MOVJ C01770 VJ=0.78
MOVL C01771 V=8.0
MOVJ C01772 VJ=0.78
MOVJ C01773 VJ=0.78
MOVJ C01774 VJ=0.78
MOVL C01775 V=8.0
MOVJ C01776 VJ=0.78
MOVJ C01777 VJ=0.78
MOVJ C01778 VJ=0.78
MOVL C01779 V=8.0
MOVJ C01780 VJ=0.78
MOVJ C01781 VJ=0.78
MOVJ C01782 VJ=0.78
MOVL C01783 V=8.0
MOVJ C01784 VJ=0.78
MOVJ C01785 VJ=0.78
MOVJ C01786 VJ=0.78
MOVL C01787 V=8.0
MOVJ C01788 VJ=0.78
MOVJ C01789 VJ=0.78
MOVJ C01790 VJ=0.78
MOVL C01791 V=8.0
MOVJ C01792 VJ=0.78
MOVJ C01793 VJ=0.78
MOVJ C01794 VJ=0.78
MOVL C01795 V=8.0
MOVJ C01796 VJ=0.78
MOVJ C01797 VJ=0.78
MOVJ C01798 VJ=0.78
MOVL C01799 V=8.0
MOVJ C01800 VJ=0.78
MOVJ C01801 VJ=0.78
MOVJ C01802 VJ=0.78
MOVL C01803 V=8.0
MOVJ C01804 VJ=0.78
MOVJ C01805 VJ=0.78
MOVJ C01806 VJ=0.78
MOVL C01807 V=8.0
MOVJ C01808 VJ=0.78
MOVJ C01809 VJ=0.78
MOVJ C01810 VJ=0.78
MOVL C01811 V=8.0
MOVJ C01812 VJ=0.78
MOVJ C01813 VJ=0.78
MOVJ C01814 VJ=0.78
MOVL C01815 V=8.0
MOVJ C01816 VJ=0.78
MOVJ C01817 VJ=0.78
MOVJ C01818 VJ=0.78
MOVL C01819 V=8.0
MOVJ C01820 VJ=0.78
MOVJ C01821 VJ=0.78
MOVJ C01822 VJ=0.78
MOVL C01823 V=8.0
MOVJ C01824 VJ=0.78
MOVJ C01825 VJ=0.78
MOVJ C01826 VJ=0.78
MOVL C01827 V=8.0
MOVJ C01828 VJ=0.78
MOVJ C01829 VJ=0.78
MOVJ C01830 VJ=0.78
MOVL C01831 V=8.0
MOVJ C01832 VJ=0.78
MOVJ C01833 VJ=0.78
MOVJ C01834 VJ=0.78
MOVL C01835 V=8.0
MOVJ C01836 VJ=0.78
MOVJ C01837 VJ=0.78
MOVJ C01838 VJ=0.78
MOVL C01839 V=8.0
MOVJ C01840 VJ=0.78
MOVJ C01841 VJ=0.78
MOVJ C01842 VJ=0.78
MOVL C01843 V=8.0
MOVJ C01844 VJ=0.78
MOVJ C01845 VJ=0.78
MOVJ C01846 VJ=0.78
MOVL C01847 V=8.0
MOVJ C01848 VJ=0.78
MOVJ C01849 VJ=0.78
MOVJ C01850 VJ=0.78
MOVL C01851 V=8.0
MOVJ C01852 VJ=0.78
MOVJ C01853 VJ=0.78
MOVJ C01854 VJ=0.78
MOVL C01855 V=8.0
MOVJ C01856 VJ=0.78
MOVJ C01857 VJ=0.78
MOVJ C01858 VJ=0.78
MOVL C01859 V=8.0
MOVJ C01860 VJ=0.78
MOVJ C01861 VJ=0.78
MOVJ C01862 VJ=0.78
MOVL C01863 V=8.0
MOVJ C01864 VJ=0.78
MOVJ C01865 VJ=0.78
MOVJ C01866 VJ=0.78
MOVL C01867 V=8.0
MOVJ C01868 VJ=0.78
MOVJ C01869 VJ=0.78
MOVJ C01870 VJ=0.78
MOVL C01871 V=8.0
MOVJ C01872 VJ=0.78
MOVJ C01873 VJ=0.78
MOVJ C01874 VJ=0.78
MOVL C01875 V=8.0
MOVJ C01876 VJ=0.78
MOVJ C01877 VJ=0.78
MOVJ C01878 VJ=0.78
MOVL C01879 V=8.0
MOVJ C01880 VJ=0.78
MOVJ C01881 VJ=0.78
MOVJ C01882 VJ=0.78
MOVL C01883 V=8.0
MOVJ C01884 VJ=0.78
MOVJ C01885 VJ=0.78
MOVJ C01886 VJ=0.78
MOVL C01887 V=8.0
MOVJ C01888 VJ=0.78
MOVJ C01889 VJ=0.78
MOVJ C01890 VJ=0.78
MOVL C01891 V=8.0
MOVJ C01892 VJ=0.78
MOVJ C01893 VJ=0.78
MOVJ C01894 VJ=0.78
MOVL C01895 V=8.0
MOVJ C01896 VJ=0.78
MOVJ C01897 VJ=0.78
MOVJ C01898 VJ=0.78
MOVL C01899 V=8.0
MOVJ C01900 VJ=0.78
MOVJ C01901 VJ=0.78
MOVJ C01902 VJ=0.78
MOVL C01903 V=8.0
MOVJ C01904 VJ=0.78
MOVJ C01905 VJ=0.78
MOVJ C01906 VJ=0.78
MOVL C01907 V=8.0
MOVJ C01908 VJ=0.78
MOVJ C01909 VJ=0.78
MOVJ C01910 VJ=0.78
MOVL C01911 V=8.0
MOVJ C01912 VJ=0.78
MOVJ C01913 VJ=0.78
MOVJ C01914 VJ=0.78
MOVL C01915 V=8.0
MOVJ C01916 VJ=0.78
MOVJ C01917 VJ=0.78
MOVJ C01918 VJ=0.78
MOVL C01919 V=8.0
MOVJ C01920 VJ=0.78
MOVJ C01921 VJ=0.78
MOVJ C01922 VJ=0.78
MOVL C01923 V=8.0
MOVJ C01924 VJ=0.78
MOVJ C01925 VJ=0.78
MOVJ C01926 VJ=0.78
MOVL C01927 V=8.0
MOVJ C01928 VJ=0.78
MOVJ C01929 VJ=0.78
MOVJ C01930 VJ=0.78
MOVL C01931 V=8.0
MOVJ C01932 VJ=0.78
MOVJ C01933 VJ=0.78
MOVJ C01934 VJ=0.78
MOVL C01935 V=8.0
MOVJ C01936 VJ=0.78
MOVJ C01937 VJ=0.78
MOVJ C01938 VJ=0.78
MOVL C01939 V=8.0
MOVJ C01940 VJ=0.78
MOVJ C01941 VJ=0.78
MOVJ C01942 VJ=0.78
MOVL C01943 V=8.0
MOVJ C01944 VJ=0.78
MOVJ C01945 VJ=0.78
MOVJ C01946 VJ=0.78
MOVL C01947 V=8.0
MOVJ C01948 VJ=0.78
MOVJ C01949 VJ=0.78
MOVJ C01950 VJ=0.78
MOVL C01951 V=8.0
MOVJ C01952 VJ=0.78
MOVJ C01953 VJ=0.78
MOVJ C01954 VJ=0.78
MOVL C01955 V=8.0
MOVJ C01956 VJ=0.78
MOVJ C01957 VJ=0.78
MOVJ C01958 VJ=0.78
MOVL C01959 V=8.0
MOVJ C01960 VJ=0.78
MOVJ C01961 VJ=0.78
MOVJ C01962 VJ=0.78
MOVL C01963 V=8.0
MOVJ C01964 VJ=0.78
MOVJ C01965 VJ=0.78
MOVJ C01966 VJ=0.78
MOVL C01967 V=8.0
MOVJ C01968 VJ=0.78
MOVJ C01969 VJ=0.78
MOVJ C01970 VJ=0.78
MOVL C01971 V=8.0
MOVJ C01972 VJ=0.78
MOVJ C01973 VJ=0.78
MOVJ C01974 VJ=0.78
MOVL C01975 V=8.0
MOVJ C01976 VJ=0.78
MOVJ C01977 VJ=0.78
MOVJ C01978 VJ=0.78
MOVL C01979 V=8.0
MOVJ C01980 VJ=0.78
MOVJ C01981 VJ=0.78
MOVJ C01982 VJ=0.78
MOVL C01983 V=8.0
MOVJ C01984 VJ=0.78
MOVJ C01985 VJ=0.78
MOVJ C01986 VJ=0.78
MOVL C01987 V=8.0
MOVJ C01988 VJ=0.78
MOVJ C01989 VJ=0.78
MOVJ C01990 VJ=0.78
MOVL C01991 V=8.0
MOVJ C01992 VJ=0.78
MOVJ C01993 VJ=0.78
MOVJ C01994 VJ=0.78
MOVL C01995 V=8.0
MOVJ C01996 VJ=0.78
MOVJ C01997 VJ=0.78
MOVJ C01998 VJ=0.78
MOVL C01999 V=8.0
MOVJ C02000 VJ=0.78
MOVJ C02001 VJ=0.78
MOVJ C02002 VJ=0.78
MOVL C02003 V=8.0
MOVJ C02004 VJ=0.78
MOVJ C02005 VJ=0.78
MOVJ C02006 VJ=0.78
MOVL C02007 V=8.0
MOVJ C02008 VJ=0.78
MOVJ C02009 VJ=0.78
MOVJ C02010 VJ=0.78
MOVL C02011 V=8.0
MOVJ C02012 VJ=0.78
MOVJ C02013 VJ=0.78
MOVJ C02014 VJ=0.78
MOVL C02015 V=8.0
MOVJ C02016 VJ=0.78
MOVJ C02017 VJ=0.78
MOVJ C02018 VJ=0.78
MOVL C02019 V=8.0
MOVJ C02020 VJ=0.78
MOVJ C02021 VJ=0.78
MOVJ C02022 VJ=0.78
MOVL C02023 V=8.0
MOVJ C02024 VJ=0.78
MOVJ C02025 VJ=0.78
MOVJ C02026 VJ=0.78
MOVL C02027 V=8.0
MOVJ C02028 VJ=0.78
MOVJ C02029 VJ=0.78
MOVJ C02030 VJ=0.78
MOVL C02031 V=8.0
MOVJ C02032 VJ=0.78
MOVJ C02033 VJ=0.78
MOVJ C02034 VJ=0.78
MOVL C02035 V=8.0
MOVJ C02036 VJ=0.78
MOVJ C02037 VJ=0.78
MOVJ C02038 VJ=0.78
MOVL C02039 V=8.0
MOVJ C02040 VJ=0.78
MOVJ C02041 VJ=0.78
MOVJ C02042 VJ=0.78
MOVL C02043 V=8.0
MOVJ C02044 VJ=0.78
MOVJ C02045 VJ=0.78
MOVJ C02046 VJ=0.78
MOVL C02047 V=8.0
MOVJ C02048 VJ=0.78
MOVJ C02049 VJ=0.78
MOVJ C02050 VJ=0.78
MOVL C02051 V=8.0
MOVJ C02052 VJ=0.78
MOVJ C02053 VJ=0.78
MOVJ C02054 VJ=0.78
MOVL C02055 V=8.0
MOVJ C02056 VJ=0.78
MOVJ C02057 VJ=0.78
MOVJ C02058 VJ=0.78
MOVL C02059 V=8.0
MOVJ C02060 VJ=0.78
MOVJ C02061 VJ=0.78
MOVJ C02062 VJ=0.78
MOVL C02063 V=8.0
MOVJ C02064 VJ=0.78
MOVJ C02065 VJ=0.78
MOVJ C02066 VJ=0.78
MOVL C02067 V=8.0
MOVJ C02068 VJ=0.78
MOVJ C02069 VJ=0.78
MOVJ C02070 VJ=0.78
MOVL C02071 V=8.0
MOVJ C02072 VJ=0.78
MOVJ C02073 VJ=0.78
MOVJ C02074 VJ=0.78
MOVL C02075 V=8.0
MOVJ C02076 VJ=0.78
MOVJ C02077 VJ=0.78
MOVJ C02078 VJ=0.78
MOVL C02079 V=8.0
MOVJ C02080 VJ=0.78
MOVJ C02081 VJ=0.78
MOVJ C02082 VJ=0.78
MOVL C02083 V=8.0
MOVJ C02084 VJ=0.78
MOVJ C02085 VJ=0.78
MOVJ C02086 VJ=0.78
MOVL C02087 V=8.0
MOVJ C02088 VJ=0.78
MOVJ C02089 VJ=0.78
MOVJ C02090 VJ=0.78
MOVL C02091 V=8.0
MOVJ C02092 VJ=0.78
MOVJ C02093 VJ=0.78
MOVJ C02094 VJ=0.78
MOVL C02095 V=8.0
MOVJ C02096 VJ=0.78
MOVJ C02097 VJ=0.78
MOVJ C02098 VJ=0.78
MOVL C02099 V=8.0
MOVJ C02100 VJ=0.78
MOVJ C02101 VJ=0.78
MOVJ C02102 VJ=0.78
MOVL C02103 V=8.0
MOVJ C02104 VJ=0.78
MOVJ C02105 VJ=0.78
MOVJ C02106 VJ=0.78
MOVL C02107 V=8.0
MOVJ C02108 VJ=0.78
MOVJ C02109 VJ=0.78
MOVJ C02110 VJ=0.78
MOVL C02111 V=8.0
MOVJ C02112 VJ=0.78
MOVJ C02113 VJ=0.78
MOVJ C02114 VJ=0.78
MOVL C02115 V=8.0
MOVJ C02116 VJ=0.78
MOVJ C02117 VJ=0.78
MOVJ C02118 VJ=0.78
MOVL C02119 V=8.0
MOVJ C02120 VJ=0.78
MOVJ C02121 VJ=0.78
MOVJ C02122 VJ=0.78
MOVL C02123 V=8.0
MOVJ C02124 VJ=0.78
MOVJ C02125 VJ=0.78
MOVJ C02126 VJ=0.78
MOVL C02127 V=8.0
MOVJ C02128 VJ=0.78
MOVJ C02129 VJ=0.78
MOVJ C02130 VJ=0.78
MOVL C02131 V=8.0
MOVJ C02132 VJ=0.78
MOVJ C02133 VJ=0.78
MOVJ C02134 VJ=0.78
MOVL C02135 V=8.0
MOVJ C02136 VJ=0.78
MOVJ C02137 VJ=0.78
MOVJ C02138 VJ=0.78
MOVL C02139 V=8.0
MOVJ C02140 VJ=0.78
MOVJ C02141 VJ=0.78
MOVJ C02142 VJ=0.78
MOVL C02143 V=8.0
MOVJ C02144 VJ=0.78
MOVJ C02145 VJ=0.78
MOVJ C02146 VJ=0.78
MOVL C02147 V=8.0
MOVJ C02148 VJ=0.78
MOVJ C02149 VJ=0.78
MOVJ C02150 VJ=0.78
MOVL C02151 V=8.0
MOVJ C02152 VJ=0.78
MOVJ C02153 VJ=0.78
MOVJ C02154 VJ=0.78
MOVL C02155 V=8.0
MOVJ C02156 VJ=0.78
MOVJ C02157 VJ=0.78
MOVJ C02158 VJ=0.78
MOVL C02159 V=8.0
MOVJ C02160 VJ=0.78
MOVJ C02161 VJ=0.78
MOVJ C02162 VJ=0.78
MOVL C02163 V=8.0
MOVJ C02164 VJ=0.78
MOVJ C02165 VJ=0.78
MOVJ C02166 VJ=0.78
MOVL C02167 V=8.0
MOVJ C02168 VJ=0.78
MOVJ C02169 VJ=0.78
MOVJ C02170 VJ=0.78
MOVL C02171 V=8.0
MOVJ C02172 VJ=0.78
MOVJ C02173 VJ=0.78
MOVJ C02174 VJ=0.78
MOVL C02175 V=8.0
MOVJ C02176 VJ=0.78
MOVJ C02177 VJ=0.78
MOVJ C02178 VJ=0.78
MOVL C02179 V=8.0
MOVJ C02180 VJ=0.78
MOVJ C02181 VJ=0.78
MOVJ C02182 VJ=0.78
MOVL C02183 V=8.0
MOVJ C02184 VJ=0.78
MOVJ C02185 VJ=0.78
MOVJ C02186 VJ=0.78
MOVL C02187 V=8.0
MOVJ C02188 VJ=0.78
MOVJ C02189 VJ=0.78
MOVJ C02190 VJ=0.78
MOVL C02191 V=8.0
MOVJ C02192 VJ=0.78
MOVJ C02193 VJ=0.78
MOVJ C02194 VJ=0.78
MOVL C02195 V=8.0
MOVJ C02196 VJ=0.78
MOVJ C02197 VJ=0.78
MOVJ C02198 VJ=0.78
MOVL C02199 V=8.0
MOVJ C02200 VJ=0.78
MOVJ C02201 VJ=0.78
MOVJ C02202 VJ=0.78
MOVL C02203 V=8.0
MOVJ C02204 VJ=0.78
MOVJ C02205 VJ=0.78
MOVJ C02206 VJ=0.78
MOVL C02207 V=8.0
MOVJ C02208 VJ=0.78
MOVJ C02209 VJ=0.78
MOVJ C02210 VJ=0.78
MOVL C02211 V=8.0
MOVJ C02212 VJ=0.78
MOVJ C02213 VJ=0.78
MOVJ C02214 VJ=0.78
MOVL C02215 V=8.0
MOVJ C02216 VJ=0.78
MOVJ C02217 VJ=0.78
MOVJ C02218 VJ=0.78
MOVL C02219 V=8.0
MOVJ C02220 VJ=0.78
MOVJ C02221 VJ=0.78
MOVJ C02222 VJ=0.78
MOVL C02223 V=8.0
MOVJ C02224 VJ=0.78
MOVJ C02225 VJ=0.78
MOVJ C02226 VJ=0.78
MOVL C02227 V=8.0
MOVJ C02228 VJ=0.78
MOVJ C02229 VJ=0.78
MOVJ C02230 VJ=0.78
MOVL C02231 V=8.0
MOVJ C02232 VJ=0.78
MOVJ C02233 VJ=0.78
MOVJ C02234 VJ=0.78
MOVL C02235 V=8.0
MOVJ C02236 VJ=0.78
MOVJ C02237 VJ=0.78
MOVJ C02238 VJ=0.78
MOVL C02239 V=8.0
MOVJ C02240 VJ=0.78
MOVJ C02241 VJ=0.78
MOVJ C02242 VJ=0.78
MOVL C02243 V=8.0
MOVJ C02244 VJ=0.78
MOVJ C02245 VJ=0.78
MOVJ C02246 VJ=0.78
MOVL C02247 V=8.0
MOVJ C02248 VJ=0.78
MOVJ C02249 VJ=0.78
MOVJ C02250 VJ=0.78
MOVL C02251 V=8.0
MOVJ C02252 VJ=0.78
MOVJ C02253 VJ=0.78
MOVJ C02254 VJ=0.78
MOVL C02255 V=8.0
MOVJ C02256 VJ=0.78
MOVJ C02257 VJ=0.78
MOVJ C02258 VJ=0.78
MOVL C02259 V=8.0
MOVJ C02260 VJ=0.78
MOVJ C02261 VJ=0.78
MOVJ C02262 VJ=0.78
MOVL C02263 V=8.0
MOVJ C02264 VJ=0.78
MOVJ C02265 VJ=0.78
MOVJ C02266 VJ=0.78
MOVL C02267 V=8.0
MOVJ C02268 VJ=0.78
MOVJ C02269 VJ=0.78
MOVJ C02270 VJ=0.78
MOVL C02271 V=8.0
MOVJ C02272 VJ=0.78
MOVJ C02273 VJ=0.78
MOVJ C02274 VJ=0.78
MOVL C02275 V=8.0
MOVJ C02276 VJ=0.78
MOVJ C02277 VJ=0.78
MOVJ C02278 VJ=0.78
MOVL C02279 V=8.0
MOVJ C02280 VJ=0.78
MOVJ C02281 VJ=0.78
MOVJ C02282 VJ=0.78
MOVL C02283 V=8.0
MOVJ C02284 VJ=0.78
MOVJ C02285 VJ=0.78
MOVJ C02286 VJ=0.78
MOVL C02287 V=8.0
MOVJ C02288 VJ=0.78
MOVJ C02289 VJ=0.78
MOVJ C02290 VJ=0.78
MOVL C02291 V=8.0
MOVJ C02292 VJ=0.78
MOVJ C02293 VJ=0.78
MOVJ C02294 VJ=0.78
MOVL C02295 V=8.0
MOVJ C02296 VJ=0.78
MOVJ C02297 VJ=0.78
MOVJ C02298 VJ=0.78
MOVL C02299 V=8.0
MOVJ C02300 VJ=0.78
MOVJ C02301 VJ=0.78
MOVJ C02302 VJ=0.78
MOVL C02303 V=8.0
MOVJ C02304 VJ=0.78
MOVJ C02305 VJ=0.78
MOVJ C02306 VJ=0.78
MOVL C02307 V=8.0
MOVJ C02308 VJ=0.78
MOVJ C02309 VJ=0.78
MOVJ C02310 VJ=0.78
MOVL C02311 V=8.0
MOVJ C02312 VJ=0.78
MOVJ C02313 VJ=0.78
MOVJ C02314 VJ=0.78
MOVL C02315 V=8.0
MOVJ C02316 VJ=0.78
MOVJ C02317 VJ=0.78
MOVJ C02318 VJ=0.78
MOVL C02319 V=8.0
MOVJ C02320 VJ=0.78
MOVJ C02321 VJ=0.78
MOVJ C02322 VJ=0.78
MOVL C02323 V=8.0
MOVJ C02324 VJ=0.78
MOVJ C02325 VJ=0.78
MOVJ C02326 VJ=0.78
MOVL C02327 V=8.0
MOVJ C02328 VJ=0.78
MOVJ C02329 VJ=0.78
MOVJ C02330 VJ=0.78
MOVL C02331 V=8.0
MOVJ C02332 VJ=0.78
MOVJ C02333 VJ=0.78
MOVJ C02334 VJ=0.78
MOVL C02335 V=8.0
MOVJ C02336 VJ=0.78
MOVJ C02337 VJ=0.78
MOVJ C02338 VJ=0.78
MOVL C02339 V=8.0
MOVJ C02340 VJ=0.78
MOVJ C02341 VJ=0.78
MOVJ C02342 VJ=0.78
MOVL C02343 V=8.0
MOVJ C02344 VJ=0.78
MOVJ C02345 VJ=0.78
MOVJ C02346 VJ=0.78
MOVL C02347 V=8.0
MOVJ C02348 VJ=0.78
MOVJ C02349 VJ=0.78
MOVJ C02350 VJ=0.78
MOVL C02351 V=8.0
MOVJ C02352 VJ=0.78
MOVJ C02353 VJ=0.78
MOVJ C02354 VJ=0.78
MOVL C02355 V=8.0
MOVJ C02356 VJ=0.78
MOVJ C02357 VJ=0.78
MOVJ C02358 VJ=0.78
MOVL C02359 V=8.0
MOVJ C02360 VJ=0.78
MOVJ C02361 VJ=0.78
MOVJ C02362 VJ=0.78
MOVL C02363 V=8.0
MOVJ C02364 VJ=0.78
MOVJ C02365 VJ=0.78
MOVJ C02366 VJ=0.78
MOVL C02367 V=8.0
MOVJ C02368 VJ=0.78
MOVJ C02369 VJ=0.78
MOVJ C02370 VJ=0.78
MOVL C02371 V=8.0
MOVJ C02372 VJ=0.78
MOVJ C02373 VJ=0.78
MOVJ C02374 VJ=0.78
MOVL C02375 V=8.0
MOVJ C02376 VJ=0.78
MOVJ C02377 VJ=0.78
MOVJ C02378 VJ=0.78
MOVL C02379 V=8.0
MOVJ C02380 VJ=0.78
MOVJ C02381 VJ=0.78
MOVJ C02382 VJ=0.78
MOVL C02383 V=8.0
MOVJ C02384 VJ=0.78
MOVJ C02385 VJ=0.78
MOVJ C02386 VJ=0.78
MOVL C02387 V=8.0
MOVJ C02388 VJ=0.78
MOVJ C02389 VJ=0.78
MOVJ C02390 VJ=0.78
MOVL C02391 V=8.0
MOVJ C02392 VJ=0.78
MOVJ C02393 VJ=0.78
MOVJ C02394 VJ=0.78
MOVL C02395 V=8.0
MOVJ C02396 VJ=0.78
MOVJ C02397 VJ=0.78
MOVJ C02398 VJ=0.78
MOVL C02399 V=8.0
MOVJ C02400 VJ=0.78
MOVJ C02401 VJ=0.78
MOVJ C02402 VJ=0.78
MOVL C02403 V=8.0
MOVJ C02404 VJ=0.78
MOVJ C02405 VJ=0.78
MOVJ C02406 VJ=0.78
MOVL C02407 V=8.0
MOVJ C02408 VJ=0.78
MOVJ C02409 VJ=0.78
MOVJ C02410 VJ=0.78
MOVL C02411 V=8.0
MOVJ C02412 VJ=0.78
MOVJ C02413 VJ=0.78
MOVJ C02414 VJ=0.78
MOVL C02415 V=8.0
MOVJ C02416 VJ=0.78
MOVJ C02417 VJ=0.78
MOVJ C02418 VJ=0.78
MOVL C02419 V=8.0
MOVJ C02420 VJ=0.78
MOVJ C02421 VJ=0.78
MOVJ C02422 VJ=0.78
MOVL C02423 V=8.0
MOVJ C02424 VJ=0.78
MOVJ C02425 VJ=0.78
MOVJ C02426 VJ=0.78
MOVL C02427 V=8.0
MOVJ C02428 VJ=0.78
MOVJ C02429 VJ=0.78
MOVJ C02430 VJ=0.78
MOVL C02431 V=8.0
MOVJ C02432 VJ=0.78
MOVJ C02433 VJ=0.78
MOVJ C02434 VJ=0.78
MOVL C02435 V=8.0
MOVJ C02436 VJ=0.78
MOVJ C02437 VJ=0.78
MOVJ C02438 VJ=0.78
MOVL C02439 V=8.0
MOVJ C02440 VJ=0.78
MOVJ C02441 VJ=0.78
MOVJ C02442 VJ=0.78
MOVL C02443 V=8.0
MOVJ C02444 VJ=0.78
MOVJ C02445 VJ=0.78
MOVJ C02446 VJ=0.78
MOVL C02447 V=8.0
MOVJ C02448 VJ=0.78
MOVJ C02449 VJ=0.78
MOVJ C02450 VJ=0.78
MOVL C02451 V=8.0
MOVJ C02452 VJ=0.78
MOVJ C02453 VJ=0.78
MOVJ C02454 VJ=0.78
MOVL C02455 V=8.0
MOVJ C02456 VJ=0.78
MOVJ C02457 VJ=0.78
MOVJ C02458 VJ=0.78
MOVL C02459 V=8.0
MOVJ C02460 VJ=0.78
MOVJ C02461 VJ=0.78
MOVJ C02462 VJ=0.78
MOVL C02463 V=8.0
MOVJ C02464 VJ=0.78
MOVJ C02465 VJ=0.78
MOVJ C02466 VJ=0.78
MOVL C02467 V=8.0
MOVJ C02468 VJ=0.78
MOVJ C02469 VJ=0.78
MOVJ C02470 VJ=0.78
MOVL C02471 V=8.0
MOVJ C02472 VJ=0.78
MOVJ C02473 VJ=0.78
MOVJ C02474 VJ=0.78
MOVL C02475 V=8.0
MOVJ C02476 VJ=0.78
MOVJ C02477 VJ=0.78
MOVJ C02478 VJ=0.78
MOVL C02479 V=8.0
MOVJ C02480 VJ=0.78
MOVJ C02481 VJ=0.78
MOVJ C02482 VJ=0.78
MOVL C02483 V=8.0
MOVJ C02484 VJ=0.78
MOVJ C02485 VJ=0.78
MOVJ C02486 VJ=0.78
MOVL C02487 V=8.0
MOVJ C02488 VJ=0.78
MOVJ C02489 VJ=0.78
MOVJ C02490 VJ=0.78
MOVL C02491 V=8.0
MOVJ C02492 VJ=0.78
MOVJ C02493 VJ=0.78
MOVJ C02494 VJ=0.78
MOVL C02495 V=8.0
MOVJ C02496 VJ=0.78
MOVJ C02497 VJ=0.78
MOVJ C02498 VJ=0.78
MOVL C02499 V=8.0
MOVJ C02500 VJ=0.78
MOVJ C02501 VJ=0.78
MOVJ C02502 VJ=0.78
MOVL C02503 V=8.0
MOVJ C02504 VJ=0.78
MOVJ C02505 VJ=0.78
MOVJ C02506 VJ=0.78
MOVL C02507 V=8.0
MOVJ C02508 VJ=0.78
MOVJ C02509 VJ=0.78
MOVJ C02510 VJ=0.78
MOVL C02511 V=8.0
MOVJ C02512 VJ=0.78
MOVJ C02513 VJ=0.78
MOVJ C02514 VJ=0.78
MOVL C02515 V=8.0
MOVJ C02516 VJ=0.78
MOVJ C02517 VJ=0.78
MOVJ C02518 VJ=0.78
MOVL C02519 V=8.0
MOVJ C02520 VJ=0.78
MOVJ C02521 VJ=0.78
MOVJ C02522 VJ=0.78
MOVL C02523 V=8.0
MOVJ C02524 VJ=0.78
MOVJ C02525 VJ=0.78
MOVJ C02526 VJ=0.78
MOVL C02527 V=8.0
MOVJ C02528 VJ=0.78
MOVJ C02529 VJ=0.78
MOVJ C02530 VJ=0.78
MOVL C02531 V=8.0
MOVJ C02532 VJ=0.78
MOVJ C02533 VJ=0.78
MOVJ C02534 VJ=0.78
MOVL C02535 V=8.0
MOVJ C02536 VJ=0.78
MOVJ C02537 VJ=0.78
MOVJ C02538 VJ=0.78
MOVL C02539 V=8.0
MOVJ C02540 VJ=0.78
MOVJ C02541 VJ=0.78
MOVJ C02542 VJ=0.78
MOVL C02543 V=8.0
MOVJ C02544 VJ=0.78
MOVJ C02545 VJ=0.78
MOVJ C02546 VJ=0.78
MOVL C02547 V=8.0
MOVJ C02548 VJ=0.78
MOVJ C02549 VJ=0.78
MOVJ C02550 VJ=0.78
MOVL C02551 V=8.0
MOVJ C02552 VJ=0.78
MOVJ C02553 VJ=0.78
MOVJ C02554 VJ=0.78
MOVL C02555 V=8.0
MOVJ C02556 VJ=0.78
MOVJ C02557 VJ=0.78
MOVJ C02558 VJ=0.78
MOVL C02559 V=8.0
MOVJ C02560 VJ=0.78
MOVJ C02561 VJ=0.78
MOVJ C02562 VJ=0.78
MOVL C02563 V=8.0
MOVJ C02564 VJ=0.78
MOVJ C02565 VJ=0.78
MOVJ C02566 VJ=0.78
MOVL C02567 V=8.0
MOVJ C02568 VJ=0.78
MOVJ C02569 VJ=0.78
MOVJ C02570 VJ=0.78
MOVL C02571 V=8.0
MOVJ C02572 VJ=0.78
MOVJ C02573 VJ=0.78
MOVJ C02574 VJ=0.78
MOVL C02575 V=8.0
MOVJ C02576 VJ=0.78
MOVJ C02577 VJ=0.78
MOVJ C02578 VJ=0.78
MOVL C02579 V=8.0
MOVJ C02580 VJ=0.78
MOVJ C02581 VJ=0.78
MOVJ C02582 VJ=0.78
MOVL C02583 V=8.0
MOVJ C02584 VJ=0.78
MOVJ C02585 VJ=0.78
MOVJ C02586 VJ=0.78
MOVL C02587 V=8.0
MOVJ C02588 VJ=0.78
MOVJ C02589 VJ=0.78
MOVJ C02590 VJ=0.78
MOVL C02591 V=8.0
MOVJ C02592 VJ=0.78
MOVJ C02593 VJ=0.78
MOVJ C02594 VJ=0.78
MOVL C02595 V=8.0
MOVJ C02596 VJ=0.78
MOVJ C02597 VJ=0.78
MOVJ C02598 VJ=0.78
MOVL C02599 V=8.0
MOVJ C02600 VJ=0.78
MOVJ C02601 VJ=0.78
MOVJ C02602 VJ=0.78
MOVL C02603 V=8.0
MOVJ C02604 VJ=0.78
MOVJ C02605 VJ=0.78
MOVJ C02606 VJ=0.78
MOVL C02607 V=8.0
MOVJ C02608 VJ=0.78
MOVJ C02609 VJ=0.78
MOVJ C02610 VJ=0.78
MOVL C02611 V=8.0
MOVJ C02612 VJ=0.78
MOVJ C02613 VJ=0.78
MOVJ C02614 VJ=0.78
MOVL C02615 V=8.0
MOVJ C02616 VJ=0.78
MOVJ C02617 VJ=0.78
MOVJ C02618 VJ=0.78
MOVL C02619 V=8.0
MOVJ C02620 VJ=0.78
MOVJ C02621 VJ=0.78
MOVJ C02622 VJ=0.78
MOVL C02623 V=8.0
MOVJ C02624 VJ=0.78
MOVJ C02625 VJ=0.78
MOVJ C02626 VJ=0.78
MOVL C02627 V=8.0
MOVJ C02628 VJ=0.78
MOVJ C02629 VJ=0.78
MOVJ C02630 VJ=0.78
MOVL C02631 V=8.0
MOVJ C02632 VJ=0.78
MOVJ C02633 VJ=0.78
MOVJ C02634 VJ=0.78
MOVL C02635 V=8.0
MOVJ C02636 VJ=0.78
MOVJ C02637 VJ=0.78
MOVJ C02638 VJ=0.78
MOVL C02639 V=8.0
MOVJ C02640 VJ=0.78
MOVJ C02641 VJ=0.78
MOVJ C02642 VJ=0.78
MOVL C02643 V=8.0
MOVJ C02644 VJ=0.78
MOVJ C02645 VJ=0.78
MOVJ C02646 VJ=0.78
MOVL C02647 V=8.0
MOVJ C02648 VJ=0.78
MOVJ C02649 VJ=0.78
MOVJ C02650 VJ=0.78
MOVL C02651 V=8.0
MOVJ C02652 VJ=0.78
MOVJ C02653 VJ=0.78
MOVJ C02654 VJ=0.78
MOVL C02655 V=8.0
MOVJ C02656 VJ=0.78
MOVJ C02657 VJ=0.78
MOVJ C02658 VJ=0.78
MOVL C02659 V=8.0
MOVJ C02660 VJ=0.78
MOVJ C02661 VJ=0.78
MOVJ C02662 VJ=0.78
MOVL C02663 V=8.0
MOVJ C02664 VJ=0.78
MOVJ C02665 VJ=0.78
MOVJ C02666 VJ=0.78
MOVL C02667 V=8.0
MOVJ C02668 VJ=0.78
MOVJ C02669 VJ=0.78
MOVJ C02670 VJ=0.78
MOVL C02671 V=8.0
MOVJ C02672 VJ=0.78
MOVJ C02673 VJ=0.78
MOVJ C02674 VJ=0.78
MOVL C02675 V=8.0
MOVJ C02676 VJ=0.78
MOVJ C02677 VJ=0.78
MOVJ C02678 VJ=0.78
MOVL C02679 V=8.0
MOVJ C02680 VJ=0.78
MOVJ C02681 VJ=0.78
MOVJ C02682 VJ=0.78
MOVL C02683 V=8.0
MOVJ C02684 VJ=0.78
MOVJ C02685 VJ=0.78
MOVJ C02686 VJ=0.78
MOVL C02687 V=8.0
MOVJ C02688 VJ=0.78
MOVJ C02689 VJ=0.78
MOVJ C02690 VJ=0.78
MOVL C02691 V=8.0
MOVJ C02692 VJ=0.78
MOVJ C02693 VJ=0.78
MOVJ C02694 VJ=0.78
MOVL C02695 V=8.0
MOVJ C02696 VJ=0.78
MOVJ C02697 VJ=0.78
MOVJ C02698 VJ=0.78
MOVL C02699 V=8.0
MOVJ C02700 VJ=0.78
MOVJ C02701 VJ=0.78
MOVJ C02702 VJ=0.78
MOVL C02703 V=8.0
MOVJ C02704 VJ=0.78
MOVJ C02705 VJ=0.78
MOVJ C02706 VJ=0.78
MOVL C02707 V=8.0
MOVJ C02708 VJ=0.78
MOVJ C02709 VJ=0.78
MOVJ C02710 VJ=0.78
MOVL C02711 V=8.0
MOVJ C02712 VJ=0.78
MOVJ C02713 VJ=0.78
MOVJ C02714 VJ=0.78
MOVL C02715 V=8.0
MOVJ C02716 VJ=0.78
MOVJ C02717 VJ=0.78
MOVJ C02718 VJ=0.78
MOVL C02719 V=8.0
MOVJ C02720 VJ=0.78
MOVJ C02721 VJ=0.78
MOVJ C02722 VJ=0.78
MOVL C02723 V=8.0
MOVJ C02724 VJ=0.78
MOVJ C02725 VJ=0.78
MOVJ C02726 VJ=0.78
MOVL C02727 V=8.0
MOVJ C02728 VJ=0.78
MOVJ C02729 VJ=0.78
MOVJ C02730 VJ=0.78
MOVL C02731 V=8.0
MOVJ C02732 VJ=0.78
MOVJ C02733 VJ=0.78
MOVJ C02734 VJ=0.78
MOVL C02735 V=8.0
MOVJ C02736 VJ=0.78
MOVJ C02737 VJ=0.78
MOVJ C02738 VJ=0.78
MOVL C02739 V=8.0
MOVJ C02740 VJ=0.78
MOVJ C02741 VJ=0.78
MOVJ C02742 VJ=0.78
MOVL C02743 V=8.0
MOVJ C02744 VJ=0.78
MOVJ C02745 VJ=0.78
MOVJ C02746 VJ=0.78
MOVL C02747 V=8.0
MOVJ C02748 VJ=0.78
MOVJ C02749 VJ=0.78
MOVJ C02750 VJ=0.78
MOVL C02751 V=8.0
MOVJ C02752 VJ=0.78
MOVJ C02753 VJ=0.78
MOVJ C02754 VJ=0.78
MOVL C02755 V=8.0
MOVJ C02756 VJ=0.78
MOVJ C02757 VJ=0.78
MOVJ C02758 VJ=0.78
MOVL C02759 V=8.0
MOVJ C02760 VJ=0.78
MOVJ C02761 VJ=0.78
MOVJ C02762 VJ=0.78
MOVL C02763 V=8.0
MOVJ C02764 VJ=0.78
MOVJ C02765 VJ=0.78
MOVJ C02766 VJ=0.78
MOVL C02767 V=8.0
MOVJ C02768 VJ=0.78
MOVJ C02769 VJ=0.78
MOVJ C02770 VJ=0.78
MOVL C02771 V=8.0
MOVJ C02772 VJ=0.78
MOVJ C02773 VJ=0.78
MOVJ C02774 VJ=0.78
MOVL C02775 V=8.0
MOVJ C02776 VJ=0.78
MOVJ C02777 VJ=0.78
MOVJ C02778 VJ=0.78
MOVL C02779 V=8.0
MOVJ C02780 VJ=0.78
MOVJ C02781 VJ=0.78
MOVJ C02782 VJ=0.78
MOVL C02783 V=8.0
MOVJ C02784 VJ=0.78
MOVJ C02785 VJ=0.78
MOVJ C02786 VJ=0.78
MOVL C02787 V=8.0
MOVJ C02788 VJ=0.78
MOVJ C02789 VJ=0.78
MOVJ C02790 VJ=0.78
MOVL C02791 V=8.0
MOVJ C02792 VJ=0.78
MOVJ C02793 VJ=0.78
MOVJ C02794 VJ=0.78
MOVL C02795 V=8.0
MOVJ C02796 VJ=0.78
MOVJ C02797 VJ=0.78
MOVJ C02798 VJ=0.78
MOVL C02799 V=8.0
MOVJ C02800 VJ=0.78
MOVJ C02801 VJ=0.78
MOVJ C02802 VJ=0.78
MOVL C02803 V=8.0
MOVJ C02804 VJ=0.78
MOVJ C02805 VJ=0.78
MOVJ C02806 VJ=0.78
MOVL C02807 V=8.0
MOVJ C02808 VJ=0.78
MOVJ C02809 VJ=0.78
MOVJ C02810 VJ=0.78
MOVL C02811 V=8.0
MOVJ C02812 VJ=0.78
MOVJ C02813 VJ=0.78
MOVJ C02814 VJ=0.78
MOVL C02815 V=8.0
MOVJ C02816 VJ=0.78
MOVJ C02817 VJ=0.78
MOVJ C02818 VJ=0.78
MOVL C02819 V=8.0
MOVJ C02820 VJ=0.78
MOVJ C02821 VJ=0.78
MOVJ C02822 VJ=0.78
MOVL C02823 V=8.0
MOVJ C02824 VJ=0.78
MOVJ C02825 VJ=0.78
MOVJ C02826 VJ=0.78
MOVL C02827 V=8.0
MOVJ C02828 VJ=0.78
MOVJ C02829 VJ=0.78
MOVJ C02830 VJ=0.78
MOVL C02831 V=8.0
MOVJ C02832 VJ=0.78
MOVJ C02833 VJ=0.78
MOVJ C02834 VJ=0.78
MOVL C02835 V=8.0
MOVJ C02836 VJ=0.78
MOVJ C02837 VJ=0.78
MOVJ C02838 VJ=0.78
MOVL C02839 V=8.0
MOVJ C02840 VJ=0.78
MOVJ C02841 VJ=0.78
MOVJ C02842 VJ=0.78
MOVL C02843 V=8.0
MOVJ C02844 VJ=0.78
MOVJ C02845 VJ=0.78
MOVJ C02846 VJ=0.78
MOVL C02847 V=8.0
MOVJ C02848 VJ=0.78
MOVJ C02849 VJ=0.78
MOVJ C02850 VJ=0.78
MOVL C02851 V=8.0
MOVJ C02852 VJ=0.78
MOVJ C02853 VJ=0.78
MOVJ C02854 VJ=0.78
MOVL C02855 V=8.0
MOVJ C02856 VJ=0.78
MOVJ C02857 VJ=0.78
MOVJ C02858 VJ=0.78
MOVL C02859 V=8.0
MOVJ C02860 VJ=0.78
MOVJ C02861 VJ=0.78
MOVJ C02862 VJ=0.78
MOVL C02863 V=8.0
MOVJ C02864 VJ=0.78
MOVJ C02865 VJ=0.78
MOVJ C02866 VJ=0.78
MOVL C02867 V=8.0
MOVJ C02868 VJ=0.78
MOVJ C02869 VJ=0.78
MOVJ C02870 VJ=0.78
MOVL C02871 V=8.0
MOVJ C02872 VJ=0.78
MOVJ C02873 VJ=0.78
MOVJ C02874 VJ=0.78
MOVL C02875 V=8.0
MOVJ C02876 VJ=0.78
MOVJ C02877 VJ=0.78
MOVJ C02878 VJ=0.78
MOVL C02879 V=8.0
MOVJ C02880 VJ=0.78
MOVJ C02881 VJ=0.78
MOVJ C02882 VJ=0.78
MOVL C02883 V=8.0
MOVJ C02884 VJ=0.78
MOVJ C02885 VJ=0.78
MOVJ C02886 VJ=0.78
MOVL C02887 V=8.0
MOVJ C02888 VJ=0.78
MOVJ C02889 VJ=0.78
MOVJ C02890 VJ=0.78
MOVL C02891 V=8.0
MOVJ C02892 VJ=0.78
MOVJ C02893 VJ=0.78
MOVJ C02894 VJ=0.78
MOVL C02895 V=8.0
MOVJ C02896 VJ=0.78
MOVJ C02897 VJ=0.78
MOVJ C02898 VJ=0.78
MOVL C02899 V=8.0
MOVJ C02900 VJ=0.78
MOVJ C02901 VJ=0.78
MOVJ C02902 VJ=0.78
MOVL C02903 V=8.0
MOVJ C02904 VJ=0.78
MOVJ C02905 VJ=0.78
MOVJ C02906 VJ=0.78
MOVL C02907 V=8.0
MOVJ C02908 VJ=0.78
MOVJ C02909 VJ=0.78
MOVJ C02910 VJ=0.78
MOVL C02911 V=8.0
MOVJ C02912 VJ=0.78
MOVJ C02913 VJ=0.78
MOVJ C02914 VJ=0.78
MOVL C02915 V=8.0
MOVJ C02916 VJ=0.78
MOVJ C02917 VJ=0.78
MOVJ C02918 VJ=0.78
MOVL C02919 V=8.0
MOVJ C02920 VJ=0.78
MOVJ C02921 VJ=0.78
MOVJ C02922 VJ=0.78
MOVL C02923 V=8.0
MOVJ C02924 VJ=0.78
MOVJ C02925 VJ=0.78
MOVJ C02926 VJ=0.78
MOVL C02927 V=8.0
MOVJ C02928 VJ=0.78
MOVJ C02929 VJ=0.78
MOVJ C02930 VJ=0.78
MOVL C02931 V=8.0
MOVJ C02932 VJ=0.78
MOVJ C02933 VJ=0.78
MOVJ C02934 VJ=0.78
MOVL C02935 V=8.0
MOVJ C02936 VJ=0.78
MOVJ C02937 VJ=0.78
MOVJ C02938 VJ=0.78
MOVL C02939 V=8.0
MOVJ C02940 VJ=0.78
MOVJ C02941 VJ=0.78
MOVJ C02942 VJ=0.78
MOVL C02943 V=8.0
MOVJ C02944 VJ=0.78
MOVJ C02945 VJ=0.78
MOVJ C02946 VJ=0.78
MOVL C02947 V=8.0
MOVJ C02948 VJ=0.78
MOVJ C02949 VJ=0.78
MOVJ C02950 VJ=0.78
MOVL C02951 V=8.0
MOVJ C02952 VJ=0.78
MOVJ C02953 VJ=0.78
MOVJ C02954 VJ=0.78
MOVL C02955 V=8.0
MOVJ C02956 VJ=0.78
MOVJ C02957 VJ=0.78
MOVJ C02958 VJ=0.78
MOVL C02959 V=8.0
MOVJ C02960 VJ=0.78
MOVJ C02961 VJ=0.78
MOVJ C02962 VJ=0.78
MOVL C02963 V=8.0
MOVJ C02964 VJ=0.78
MOVJ C02965 VJ=0.78
MOVJ C02966 VJ=0.78
MOVL C02967 V=8.0
MOVJ C02968 VJ=0.78
MOVJ C02969 VJ=0.78
MOVJ C02970 VJ=0.78
MOVL C02971 V=8.0
MOVJ C02972 VJ=0.78
MOVJ C02973 VJ=0.78
MOVJ C02974 VJ=0.78
MOVL C02975 V=8.0
MOVJ C02976 VJ=0.78
MOVJ C02977 VJ=0.78
MOVJ C02978 VJ=0.78
MOVL C02979 V=8.0
MOVJ C02980 VJ=0.78
MOVJ C02981 VJ=0.78
MOVJ C02982 VJ=0.78
MOVL C02983 V=8.0
MOVJ C02984 VJ=0.78
MOVJ C02985 VJ=0.78
MOVJ C02986 VJ=0.78
MOVL C02987 V=8.0
MOVJ C02988 VJ=0.78
MOVJ C02989 VJ=0.78
MOVJ C02990 VJ=0.78
MOVL C02991 V=8.0
MOVJ C02992 VJ=0.78
MOVJ C02993 VJ=0.78
MOVJ C02994 VJ=0.78
MOVL C02995 V=8.0
MOVJ C02996 VJ=0.78
MOVJ C02997 VJ=0.78
MOVJ C02998 VJ=0.78
MOVL C02999 V=8.0
MOVJ C03000 VJ=0.78
MOVJ C03001 VJ=0.78
MOVJ C03002 VJ=0.78
MOVL C03003 V=8.0
MOVJ C03004 VJ=0.78
MOVJ C03005 VJ=0.78
MOVJ C03006 VJ=0.78
MOVL C03007 V=8.0
MOVJ C03008 VJ=0.78
MOVJ C03009 VJ=0.78
MOVJ C03010 VJ=0.78
MOVL C03011 V=8.0
MOVJ C03012 VJ=0.78
MOVJ C03013 VJ=0.78
MOVJ C03014 VJ=0.78
MOVL C03015 V=8.0
MOVJ C03016 VJ=0.78
MOVJ C03017 VJ=0.78
MOVJ C03018 VJ=0.78
MOVL C03019 V=8.0
MOVJ C03020 VJ=0.78
MOVJ C03021 VJ=0.78
MOVJ C03022 VJ=0.78
MOVL C03023 V=8.0
MOVJ C03024 VJ=0.78
MOVJ C03025 VJ=0.78
MOVJ C03026 VJ=0.78
MOVL C03027 V=8.0
MOVJ C03028 VJ=0.78
MOVJ C03029 VJ=0.78
MOVJ C03030 VJ=0.78
MOVL C03031 V=8.0
MOVJ C03032 VJ=0.78
MOVJ C03033 VJ=0.78
MOVJ C03034 VJ=0.78
MOVL C03035 V=8.0
MOVJ C03036 VJ=0.78
MOVJ C03037 VJ=0.78
MOVJ C03038 VJ=0.78
MOVL C03039 V=8.0
MOVJ C03040 VJ=0.78
MOVJ C03041 VJ=0.78
MOVJ C03042 VJ=0.78
MOVL C03043 V=8.0
MOVJ C03044 VJ=0.78
MOVJ C03045 VJ=0.78
MOVJ C03046 VJ=0.78
MOVL C03047 V=8.0
MOVJ C03048 VJ=0.78
MOVJ C03049 VJ=0.78
MOVJ C03050 VJ=0.78
MOVL C03051 V=8.0
MOVJ C03052 VJ=0.78
MOVJ C03053 VJ=0.78
MOVJ C03054 VJ=0.78
MOVL C03055 V=8.0
MOVJ C03056 VJ=0.78
MOVJ C03057 VJ=0.78
MOVJ C03058 VJ=0.78
MOVL C03059 V=8.0
MOVJ C03060 VJ=0.78
MOVJ C03061 VJ=0.78
MOVJ C03062 VJ=0.78
MOVL C03063 V=8.0
MOVJ C03064 VJ=0.78
MOVJ C03065 VJ=0.78
MOVJ C03066 VJ=0.78
MOVL C03067 V=8.0
MOVJ C03068 VJ=0.78
MOVJ C03069 VJ=0.78
MOVJ C03070 VJ=0.78
MOVL C03071 V=8.0
MOVJ C03072 VJ=0.78
MOVJ C03073 VJ=0.78
MOVJ C03074 VJ=0.78
MOVL C03075 V=8.0
MOVJ C03076 VJ=0.78
MOVJ C03077 VJ=0.78
MOVJ C03078 VJ=0.78
MOVL C03079 V=8.0
MOVJ C03080 VJ=0.78
MOVJ C03081 VJ=0.78
MOVJ C03082 VJ=0.78
MOVL C03083 V=8.0
MOVJ C03084 VJ=0.78
MOVJ C03085 VJ=0.78
MOVJ C03086 VJ=0.78
MOVL C03087 V=8.0
MOVJ C03088 VJ=0.78
MOVJ C03089 VJ=0.78
MOVJ C03090 VJ=0.78
MOVL C03091 V=8.0
MOVJ C03092 VJ=0.78
MOVJ C03093 VJ=0.78
MOVJ C03094 VJ=0.78
MOVL C03095 V=8.0
MOVJ C03096 VJ=0.78
MOVJ C03097 VJ=0.78
MOVJ C03098 VJ=0.78
MOVL C03099 V=8.0
MOVJ C03100 VJ=0.78
MOVJ C03101 VJ=0.78
MOVJ C03102 VJ=0.78
MOVL C03103 V=8.0
MOVJ C03104 VJ=0.78
MOVJ C03105 VJ=0.78
MOVJ C03106 VJ=0.78
MOVL C03107 V=8.0
MOVJ C03108 VJ=0.78
MOVJ C03109 VJ=0.78
MOVJ C03110 VJ=0.78
MOVL C03111 V=8.0
MOVJ C03112 VJ=0.78
MOVJ C03113 VJ=0.78
MOVJ C03114 VJ=0.78
MOVL C03115 V=8.0
MOVJ C03116 VJ=0.78
MOVJ C03117 VJ=0.78
MOVJ C03118 VJ=0.78
MOVL C03119 V=8.0
MOVJ C03120 VJ=0.78
MOVJ C03121 VJ=0.78
MOVJ C03122 VJ=0.78
MOVL C03123 V=8.0
MOVJ C03124 VJ=0.78
MOVJ C03125 VJ=0.78
MOVJ C03126 VJ=0.78
MOVL C03127 V=8.0
MOVJ C03128 VJ=0.78
MOVJ C03129 VJ=0.78
MOVJ C03130 VJ=0.78
MOVL C03131 V=8.0
MOVJ C03132 VJ=0.78
MOVJ C03133 VJ=0.78
MOVJ C03134 VJ=0.78
MOVL C03135 V=8.0
MOVJ C03136 VJ=0.78
MOVJ C03137 VJ=0.78
MOVJ C03138 VJ=0.78
MOVL C03139 V=8.0
MOVJ C03140 VJ=0.78
MOVJ C03141 VJ=0.78
MOVJ C03142 VJ=0.78
MOVL C03143 V=8.0
MOVJ C03144 VJ=0.78
MOVJ C03145 VJ=0.78
MOVJ C03146 VJ=0.78
MOVL C03147 V=8.0
MOVJ C03148 VJ=0.78
MOVJ C03149 VJ=0.78
MOVJ C03150 VJ=0.78
MOVL C03151 V=8.0
MOVJ C03152 VJ=0.78
MOVJ C03153 VJ=0.78
MOVJ C03154 VJ=0.78
MOVL C03155 V=8.0
MOVJ C03156 VJ=0.78
MOVJ C03157 VJ=0.78
MOVJ C03158 VJ=0.78
MOVL C03159 V=8.0
MOVJ C03160 VJ=0.78
MOVJ C03161 VJ=0.78
MOVJ C03162 VJ=0.78
MOVL C03163 V=8.0
MOVJ C03164 VJ=0.78
MOVJ C03165 VJ=0.78
MOVJ C03166 VJ=0.78
MOVL C03167 V=8.0
MOVJ C03168 VJ=0.78
MOVJ C03169 VJ=0.78
MOVJ C03170 VJ=0.78
MOVL C03171 V=8.0
MOVJ C03172 VJ=0.78
MOVJ C03173 VJ=0.78
MOVJ C03174 VJ=0.78
MOVL C03175 V=8.0
MOVJ C03176 VJ=0.78
MOVJ C03177 VJ=0.78
MOVJ C03178 VJ=0.78
MOVL C03179 V=8.0
MOVJ C03180 VJ=0.78
MOVJ C03181 VJ=0.78
MOVJ C03182 VJ=0.78
MOVL C03183 V=8.0
MOVJ C03184 VJ=0.78
MOVJ C03185 VJ=0.78
MOVJ C03186 VJ=0.78
MOVL C03187 V=8.0
MOVJ C03188 VJ=0.78
MOVJ C03189 VJ=0.78
MOVJ C03190 VJ=0.78
MOVL C03191 V=8.0
MOVJ C03192 VJ=0.78
MOVJ C03193 VJ=0.78
MOVJ C03194 VJ=0.78
MOVL C03195 V=8.0
MOVJ C03196 VJ=0.78
MOVJ C03197 VJ=0.78
MOVJ C03198 VJ=0.78
MOVL C03199 V=8.0
MOVJ C03200 VJ=0.78
MOVJ C03201 VJ=0.78
MOVJ C03202 VJ=0.78
MOVL C03203 V=8.0
MOVJ C03204 VJ=0.78
MOVJ C03205 VJ=0.78
MOVJ C03206 VJ=0.78
MOVL C03207 V=8.0
MOVJ C03208 VJ=0.78
MOVJ C03209 VJ=0.78
MOVJ C03210 VJ=0.78
MOVL C03211 V=8.0
MOVJ C03212 VJ=0.78
MOVJ C03213 VJ=0.78
MOVJ C03214 VJ=0.78
MOVL C03215 V=8.0
MOVJ C03216 VJ=0.78
MOVJ C03217 VJ=0.78
MOVJ C03218 VJ=0.78
MOVL C03219 V=8.0
MOVJ C03220 VJ=0.78
MOVJ C03221 VJ=0.78
MOVJ C03222 VJ=0.78
MOVL C03223 V=8.0
MOVJ C03224 VJ=0.78
MOVJ C03225 VJ=0.78
MOVJ C03226 VJ=0.78
MOVL C03227 V=8.0
MOVJ C03228 VJ=0.78
MOVJ C03229 VJ=0.78
MOVJ C03230 VJ=0.78
MOVL C03231 V=8.0
MOVJ C03232 VJ=0.78
MOVJ C03233 VJ=0.78
MOVJ C03234 VJ=0.78
MOVL C03235 V=8.0
MOVJ C03236 VJ=0.78
MOVJ C03237 VJ=0.78
MOVJ C03238 VJ=0.78
MOVL C03239 V=8.0
MOVJ C03240 VJ=0.78
MOVJ C03241 VJ=0.78
MOVJ C03242 VJ=0.78
MOVL C03243 V=8.0
MOVJ C03244 VJ=0.78
MOVJ C03245 VJ=0.78
MOVJ C03246 VJ=0.78
MOVL C03247 V=8.0
MOVJ C03248 VJ=0.78
MOVJ C03249 VJ=0.78
MOVJ C03250 VJ=0.78
MOVL C03251 V=8.0
MOVJ C03252 VJ=0.78
MOVJ C03253 VJ=0.78
MOVJ C03254 VJ=0.78
MOVL C03255 V=8.0
MOVJ C03256 VJ=0.78
MOVJ C03257 VJ=0.78
MOVJ C03258 VJ=0.78
MOVL C03259 V=8.0
MOVJ C03260 VJ=0.78
MOVJ C03261 VJ=0.78
MOVJ C03262 VJ=0.78
MOVL C03263 V=8.0
MOVJ C03264 VJ=0.78
MOVJ C03265 VJ=0.78
MOVJ C03266 VJ=0.78
MOVL C03267 V=8.0
MOVJ C03268 VJ=0.78
MOVJ C03269 VJ=0.78
MOVJ C03270 VJ=0.78
MOVL C03271 V=8.0
MOVJ C03272 VJ=0.78
MOVJ C03273 VJ=0.78
MOVJ C03274 VJ=0.78
MOVL C03275 V=8.0
MOVJ C03276 VJ=0.78
MOVJ C03277 VJ=0.78
MOVJ C03278 VJ=0.78
MOVL C03279 V=8.0
MOVJ C03280 VJ=0.78
MOVJ C03281 VJ=0.78
MOVJ C03282 VJ=0.78
MOVL C03283 V=8.0
MOVJ C03284 VJ=0.78
MOVJ C03285 VJ=0.78
MOVJ C03286 VJ=0.78
MOVL C03287 V=8.0
MOVJ C03288 VJ=0.78
MOVJ C03289 VJ=0.78
MOVJ C03290 VJ=0.78
MOVL C03291 V=8.0
MOVJ C03292 VJ=0.78
MOVJ C03293 VJ=0.78
MOVJ C03294 VJ=0.78
MOVL C03295 V=8.0
MOVJ C03296 VJ=0.78
MOVJ C03297 VJ=0.78
MOVJ C03298 VJ=0.78
MOVL C03299 V=8.0
MOVJ C03300 VJ=0.78
MOVJ C03301 VJ=0.78
MOVJ C03302 VJ=0.78
MOVL C03303 V=8.0
MOVJ C03304 VJ=0.78
MOVJ C03305 VJ=0.78
MOVJ C03306 VJ=0.78
MOVL C03307 V=8.0
MOVJ C03308 VJ=0.78
MOVJ C03309 VJ=0.78
MOVJ C03310 VJ=0.78
MOVL C03311 V=8.0
MOVJ C03312 VJ=0.78
MOVJ C03313 VJ=0.78
MOVJ C03314 VJ=0.78
MOVL C03315 V=8.0
MOVJ C03316 VJ=0.78
MOVJ C03317 VJ=0.78
MOVJ C03318 VJ=0.78
MOVL C03319 V=8.0
MOVJ C03320 VJ=0.78
MOVJ C03321 VJ=0.78
MOVJ C03322 VJ=0.78
MOVL C03323 V=8.0
MOVJ C03324 VJ=0.78
MOVJ C03325 VJ=0.78
MOVJ C03326 VJ=0.78
MOVL C03327 V=8.0
MOVJ C03328 VJ=0.78
MOVJ C03329 VJ=0.78
MOVJ C03330 VJ=0.78
MOVL C03331 V=8.0
MOVJ C03332 VJ=0.78
MOVJ C03333 VJ=0.78
MOVJ C03334 VJ=0.78
MOVL C03335 V=8.0
MOVJ C03336 VJ=0.78
MOVJ C03337 VJ=0.78
MOVJ C03338 VJ=0.78
MOVL C03339 V=8.0
MOVJ C03340 VJ=0.78
MOVJ C03341 VJ=0.78
MOVJ C03342 VJ=0.78
MOVL C03343 V=8.0
MOVJ C03344 VJ=0.78
MOVJ C03345 VJ=0.78
MOVJ C03346 VJ=0.78
MOVL C03347 V=8.0
MOVJ C03348 VJ=0.78
MOVJ C03349 VJ=0.78
MOVJ C03350 VJ=0.78
MOVL C03351 V=8.0
MOVJ C03352 VJ=0.78
MOVJ C03353 VJ=0.78
MOVJ C03354 VJ=0.78
MOVL C03355 V=8.0
MOVJ C03356 VJ=0.78
MOVJ C03357 VJ=0.78
MOVJ C03358 VJ=0.78
MOVL C03359 V=8.0
MOVJ C03360 VJ=0.78
MOVJ C03361 VJ=0.78
MOVJ C03362 VJ=0.78
MOVL C03363 V=8.0
MOVJ C03364 VJ=0.78
MOVJ C03365 VJ=0.78
MOVJ C03366 VJ=0.78
MOVL C03367 V=8.0
MOVJ C03368 VJ=0.78
MOVJ C03369 VJ=0.78
MOVJ C03370 VJ=0.78
MOVL C03371 V=8.0
MOVJ C03372 VJ=0.78
MOVJ C03373 VJ=0.78
MOVJ C03374 VJ=0.78
MOVL C03375 V=8.0
MOVJ C03376 VJ=0.78
MOVJ C03377 VJ=0.78
MOVJ C03378 VJ=0.78
MOVL C03379 V=8.0
MOVJ C03380 VJ=0.78
MOVJ C03381 VJ=0.78
MOVJ C03382 VJ=0.78
MOVL C03383 V=8.0
MOVJ C03384 VJ=0.78
MOVJ C03385 VJ=0.78
MOVJ C03386 VJ=0.78
MOVL C03387 V=8.0
MOVJ C03388 VJ=0.78
MOVJ C03389 VJ=0.78
MOVJ C03390 VJ=0.78
MOVL C03391 V=8.0
MOVJ C03392 VJ=0.78
MOVJ C03393 VJ=0.78
MOVJ C03394 VJ=0.78
MOVL C03395 V=8.0
MOVJ C03396 VJ=0.78
MOVJ C03397 VJ=0.78
MOVJ C03398 VJ=0.78
MOVL C03399 V=8.0
MOVJ C03400 VJ=0.78
MOVJ C03401 VJ=0.78
MOVJ C03402 VJ=0.78
MOVL C03403 V=8.0
MOVJ C03404 VJ=0.78
MOVJ C03405 VJ=0.78
MOVJ C03406 VJ=0.78
MOVL C03407 V=8.0
MOVJ C03408 VJ=0.78
MOVJ C03409 VJ=0.78
MOVJ C03410 VJ=0.78
MOVL C03411 V=8.0
MOVJ C03412 VJ=0.78
MOVJ C03413 VJ=0.78
MOVJ C03414 VJ=0.78
MOVL C03415 V=8.0
MOVJ C03416 VJ=0.78
MOVJ C03417 VJ=0.78
MOVJ C03418 VJ=0.78
MOVL C03419 V=8.0
MOVJ C03420 VJ=0.78
MOVJ C03421 VJ=0.78
MOVJ C03422 VJ=0.78
MOVL C03423 V=8.0
MOVJ C03424 VJ=0.78
MOVJ C03425 VJ=0.78
MOVJ C03426 VJ=0.78
MOVL C03427 V=8.0
MOVJ C03428 VJ=0.78
MOVJ C03429 VJ=0.78
MOVJ C03430 VJ=0.78
MOVL C03431 V=8.0
MOVJ C03432 VJ=0.78
MOVJ C03433 VJ=0.78
MOVJ C03434 VJ=0.78
MOVL C03435 V=8.0
MOVJ C03436 VJ=0.78
MOVJ C03437 VJ=0.78
MOVJ C03438 VJ=0.78
MOVL C03439 V=8.0
MOVJ C03440 VJ=0.78
MOVJ C03441 VJ=0.78
MOVJ C03442 VJ=0.78
MOVL C03443 V=8.0
MOVJ C03444 VJ=0.78
MOVJ C03445 VJ=0.78
MOVJ C03446 VJ=0.78
MOVL C03447 V=8.0
MOVJ C03448 VJ=0.78
MOVJ C03449 VJ=0.78
MOVJ C03450 VJ=0.78
MOVL C03451 V=8.0
MOVJ C03452 VJ=0.78
MOVJ C03453 VJ=0.78
MOVJ C03454 VJ=0.78
MOVL C03455 V=8.0
MOVJ C03456 VJ=0.78
MOVJ C03457 VJ=0.78
MOVJ C03458 VJ=0.78
MOVL C03459 V=8.0
MOVJ C03460 VJ=0.78
MOVJ C03461 VJ=0.78
MOVJ C03462 VJ=0.78
MOVL C03463 V=8.0
MOVJ C03464 VJ=0.78
MOVJ C03465 VJ=0.78
MOVJ C03466 VJ=0.78
MOVL C03467 V=8.0
MOVJ C03468 VJ=0.78
MOVJ C03469 VJ=0.78
MOVJ C03470 VJ=0.78
MOVL C03471 V=8.0
MOVJ C03472 VJ=0.78
MOVJ C03473 VJ=0.78
MOVJ C03474 VJ=0.78
MOVL C03475 V=8.0
MOVJ C03476 VJ=0.78
MOVJ C03477 VJ=0.78
MOVJ C03478 VJ=0.78
MOVL C03479 V=8.0
MOVJ C03480 VJ=0.78
MOVJ C03481 VJ=0.78
MOVJ C03482 VJ=0.78
MOVL C03483 V=8.0
MOVJ C03484 VJ=0.78
MOVJ C03485 VJ=0.78
MOVJ C03486 VJ=0.78
MOVL C03487 V=8.0
MOVJ C03488 VJ=0.78
MOVJ C03489 VJ=0.78
MOVJ C03490 VJ=0.78
MOVL C03491 V=8.0
MOVJ C03492 VJ=0.78
MOVJ C03493 VJ=0.78
MOVJ C03494 VJ=0.78
MOVL C03495 V=8.0
MOVJ C03496 VJ=0.78
MOVJ C03497 VJ=0.78
MOVJ C03498 VJ=0.78
MOVL C03499 V=8.0
MOVJ C03500 VJ=0.78
MOVJ C03501 VJ=0.78
MOVJ C03502 VJ=0.78
MOVL C03503 V=8.0
MOVJ C03504 VJ=0.78
MOVJ C03505 VJ=0.78
MOVJ C03506 VJ=0.78
MOVL C03507 V=8.0
MOVJ C03508 VJ=0.78
MOVJ C03509 VJ=0.78
MOVJ C03510 VJ=0.78
MOVL C03511 V=8.0
MOVJ C03512 VJ=0.78
MOVJ C03513 VJ=0.78
MOVJ C03514 VJ=0.78
MOVL C03515 V=8.0
MOVJ C03516 VJ=0.78
MOVJ C03517 VJ=0.78
MOVJ C03518 VJ=0.78
MOVL C03519 V=8.0
MOVJ C03520 VJ=0.78
MOVJ C03521 VJ=0.78
MOVJ C03522 VJ=0.78
MOVL C03523 V=8.0
MOVJ C03524 VJ=0.78
MOVJ C03525 VJ=0.78
MOVJ C03526 VJ=0.78
MOVL C03527 V=8.0
MOVJ C03528 VJ=0.78
MOVJ C03529 VJ=0.78
MOVJ C03530 VJ=0.78
MOVL C03531 V=8.0
MOVJ C03532 VJ=0.78
MOVJ C03533 VJ=0.78
MOVJ C03534 VJ=0.78
MOVL C03535 V=8.0
MOVJ C03536 VJ=0.78
MOVJ C03537 VJ=0.78
MOVJ C03538 VJ=0.78
MOVL C03539 V=8.0
MOVJ C03540 VJ=0.78
MOVJ C03541 VJ=0.78
MOVJ C03542 VJ=0.78
MOVL C03543 V=8.0
MOVJ C03544 VJ=0.78
MOVJ C03545 VJ=0.78
MOVJ C03546 VJ=0.78
MOVL C03547 V=8.0
MOVJ C03548 VJ=0.78
MOVJ C03549 VJ=0.78
MOVJ C03550 VJ=0.78
MOVL C03551 V=8.0
MOVJ C03552 VJ=0.78
MOVJ C03553 VJ=0.78
MOVJ C03554 VJ=0.78
MOVL C03555 V=8.0
MOVJ C03556 VJ=0.78
MOVJ C03557 VJ=0.78
MOVJ C03558 VJ=0.78
MOVL C03559 V=8.0
MOVJ C03560 VJ=0.78
MOVJ C03561 VJ=0.78
MOVJ C03562 VJ=0.78
MOVL C03563 V=8.0
MOVJ C03564 VJ=0.78
MOVJ C03565 VJ=0.78
MOVJ C03566 VJ=0.78
MOVL C03567 V=8.0
MOVJ C03568 VJ=0.78
MOVJ C03569 VJ=0.78
MOVJ C03570 VJ=0.78
MOVL C03571 V=8.0
MOVJ C03572 VJ=0.78
MOVJ C03573 VJ=0.78
MOVJ C03574 VJ=0.78
MOVL C03575 V=8.0
MOVJ C03576 VJ=0.78
MOVJ C03577 VJ=0.78
MOVJ C03578 VJ=0.78
MOVL C03579 V=8.0
MOVJ C03580 VJ=0.78
MOVJ C03581 VJ=0.78
MOVJ C03582 VJ=0.78
MOVL C03583 V=8.0
MOVJ C03584 VJ=0.78
MOVJ C03585 VJ=0.78
MOVJ C03586 VJ=0.78
MOVL C03587 V=8.0
MOVJ C03588 VJ=0.78
MOVJ C03589 VJ=0.78
MOVJ C03590 VJ=0.78
MOVL C03591 V=8.0
MOVJ C03592 VJ=0.78
MOVJ C03593 VJ=0.78
MOVJ C03594 VJ=0.78
MOVL C03595 V=8.0
MOVJ C03596 VJ=0.78
MOVJ C03597 VJ=0.78
MOVJ C03598 VJ=0.78
MOVL C03599 V=8.0
MOVJ C03600 VJ=0.78
MOVJ C03601 VJ=0.78
MOVJ C03602 VJ=0.78
MOVL C03603 V=8.0
MOVJ C03604 VJ=0.78
MOVJ C03605 VJ=0.78
MOVJ C03606 VJ=0.78
MOVL C03607 V=8.0
MOVJ C03608 VJ=0.78
MOVJ C03609 VJ=0.78
MOVJ C03610 VJ=0.78
MOVL C03611 V=8.0
MOVJ C03612 VJ=0.78
MOVJ C03613 VJ=0.78
MOVJ C03614 VJ=0.78
MOVL C03615 V=8.0
MOVJ C03616 VJ=0.78
MOVJ C03617 VJ=0.78
MOVJ C03618 VJ=0.78
MOVL C03619 V=8.0
MOVJ C03620 VJ=0.78
MOVJ C03621 VJ=0.78
MOVJ C03622 VJ=0.78
MOVL C03623 V=8.0
MOVJ C03624 VJ=0.78
MOVJ C03625 VJ=0.78
MOVJ C03626 VJ=0.78
MOVL C03627 V=8.0
MOVJ C03628 VJ=0.78
MOVJ C03629 VJ=0.78
MOVJ C03630 VJ=0.78
MOVL C03631 V=8.0
MOVJ C03632 VJ=0.78
MOVJ C03633 VJ=0.78
MOVJ C03634 VJ=0.78
MOVL C03635 V=8.0
MOVJ C03636 VJ=0.78
MOVJ C03637 VJ=0.78
MOVJ C03638 VJ=0.78
MOVL C03639 V=8.0
MOVJ C03640 VJ=0.78
MOVJ C03641 VJ=0.78
MOVJ C03642 VJ=0.78
MOVL C03643 V=8.0
MOVJ C03644 VJ=0.78
MOVJ C03645 VJ=0.78
MOVJ C03646 VJ=0.78
MOVL C03647 V=8.0
MOVJ C03648 VJ=0.78
MOVJ C03649 VJ=0.78
MOVJ C03650 VJ=0.78
MOVL C03651 V=8.0
MOVJ C03652 VJ=0.78
MOVJ C03653 VJ=0.78
MOVJ C03654 VJ=0.78
MOVL C03655 V=8.0
MOVJ C03656 VJ=0.78
MOVJ C03657 VJ=0.78
MOVJ C03658 VJ=0.78
MOVL C03659 V=8.0
MOVJ C03660 VJ=0.78
MOVJ C03661 VJ=0.78
MOVJ C03662 VJ=0.78
MOVL C03663 V=8.0
MOVJ C03664 VJ=0.78
MOVJ C03665 VJ=0.78
MOVJ C03666 VJ=0.78
MOVL C03667 V=8.0
MOVJ C03668 VJ=0.78
MOVJ C03669 VJ=0.78
MOVJ C03670 VJ=0.78
MOVL C03671 V=8.0
MOVJ C03672 VJ=0.78
MOVJ C03673 VJ=0.78
MOVJ C03674 VJ=0.78
MOVL C03675 V=8.0
MOVJ C03676 VJ=0.78
MOVJ C03677 VJ=0.78
MOVJ C03678 VJ=0.78
MOVL C03679 V=8.0
MOVJ C03680 VJ=0.78
MOVJ C03681 VJ=0.78
MOVJ C03682 VJ=0.78
MOVL C03683 V=8.0
MOVJ C03684 VJ=0.78
MOVJ C03685 VJ=0.78
MOVJ C03686 VJ=0.78
MOVL C03687 V=8.0
MOVJ C03688 VJ=0.78
MOVJ C03689 VJ=0.78
MOVJ C03690 VJ=0.78
MOVL C03691 V=8.0
MOVJ C03692 VJ=0.78
MOVJ C03693 VJ=0.78
MOVJ C03694 VJ=0.78
MOVL C03695 V=8.0
MOVJ C03696 VJ=0.78
MOVJ C03697 VJ=0.78
MOVJ C03698 VJ=0.78
MOVL C03699 V=8.0
MOVJ C03700 VJ=0.78
MOVJ C03701 VJ=0.78
MOVJ C03702 VJ=0.78
MOVL C03703 V=8.0
MOVJ C03704 VJ=0.78
MOVJ C03705 VJ=0.78
MOVJ C03706 VJ=0.78
MOVL C03707 V=8.0
MOVJ C03708 VJ=0.78
MOVJ C03709 VJ=0.78
MOVJ C03710 VJ=0.78
MOVL C03711 V=8.0
MOVJ C03712 VJ=0.78
MOVJ C03713 VJ=0.78
MOVJ C03714 VJ=0.78
MOVL C03715 V=8.0
MOVJ C03716 VJ=0.78
MOVJ C03717 VJ=0.78
MOVJ C03718 VJ=0.78
MOVL C03719 V=8.0
MOVJ C03720 VJ=0.78
MOVJ C03721 VJ=0.78
MOVJ C03722 VJ=0.78
MOVL C03723 V=8.0
MOVJ C03724 VJ=0.78
MOVJ C03725 VJ=0.78
MOVJ C03726 VJ=0.78
MOVL C03727 V=8.0
MOVJ C03728 VJ=0.78
MOVJ C03729 VJ=0.78
MOVJ C03730 VJ=0.78
MOVL C03731 V=8.0
MOVJ C03732 VJ=0.78
MOVJ C03733 VJ=0.78
MOVJ C03734 VJ=0.78
MOVL C03735 V=8.0
MOVJ C03736 VJ=0.78
MOVJ C03737 VJ=0.78
MOVJ C03738 VJ=0.78
MOVL C03739 V=8.0
MOVJ C03740 VJ=0.78
MOVJ C03741 VJ=0.78
MOVJ C03742 VJ=0.78
MOVL C03743 V=8.0
MOVJ C03744 VJ=0.78
MOVJ C03745 VJ=0.78
MOVJ C03746 VJ=0.78
MOVL C03747 V=8.0
MOVJ C03748 VJ=0.78
MOVJ C03749 VJ=0.78
MOVJ C03750 VJ=0.78
MOVL C03751 V=8.0
MOVJ C03752 VJ=0.78
MOVJ C03753 VJ=0.78
MOVJ C03754 VJ=0.78
MOVL C03755 V=8.0
MOVJ C03756 VJ=0.78
MOVJ C03757 VJ=0.78
MOVJ C03758 VJ=0.78
MOVL C03759 V=8.0
MOVJ C03760 VJ=0.78
MOVJ C03761 VJ=0.78
MOVJ C03762 VJ=0.78
MOVL C03763 V=8.0
MOVJ C03764 VJ=0.78
MOVJ C03765 VJ=0.78
MOVJ C03766 VJ=0.78
MOVL C03767 V=8.0
MOVJ C03768 VJ=0.78
MOVJ C03769 VJ=0.78
MOVJ C03770 VJ=0.78
MOVL C03771 V=8.0
MOVJ C03772 VJ=0.78
MOVJ C03773 VJ=0.78
MOVJ C03774 VJ=0.78
MOVL C03775 V=8.0
MOVJ C03776 VJ=0.78
MOVJ C03777 VJ=0.78
MOVJ C03778 VJ=0.78
MOVL C03779 V=8.0
MOVJ C03780 VJ=0.78
MOVJ C03781 VJ=0.78
MOVJ C03782 VJ=0.78
MOVL C03783 V=8.0
MOVJ C03784 VJ=0.78
MOVJ C03785 VJ=0.78
MOVJ C03786 VJ=0.78
MOVL C03787 V=8.0
MOVJ C03788 VJ=0.78
MOVJ C03789 VJ=0.78
MOVJ C03790 VJ=0.78
MOVL C03791 V=8.0
MOVJ C03792 VJ=0.78
MOVJ C03793 VJ=0.78
MOVJ C03794 VJ=0.78
MOVL C03795 V=8.0
MOVJ C03796 VJ=0.78
MOVJ C03797 VJ=0.78
MOVJ C03798 VJ=0.78
MOVL C03799 V=8.0
MOVJ C03800 VJ=0.78
MOVJ C03801 VJ=0.78
MOVJ C03802 VJ=0.78
MOVL C03803 V=8.0
MOVJ C03804 VJ=0.78
MOVJ C03805 VJ=0.78
MOVJ C03806 VJ=0.78
MOVL C03807 V=8.0
MOVJ C03808 VJ=0.78
MOVJ C03809 VJ=0.78
MOVJ C03810 VJ=0.78
MOVL C03811 V=8.0
MOVJ C03812 VJ=0.78
MOVJ C03813 VJ=0.78
MOVJ C03814 VJ=0.78
MOVL C03815 V=8.0
MOVJ C03816 VJ=0.78
MOVJ C03817 VJ=0.78
MOVJ C03818 VJ=0.78
MOVL C03819 V=8.0
MOVJ C03820 VJ=0.78
MOVJ C03821 VJ=0.78
MOVJ C03822 VJ=0.78
MOVL C03823 V=8.0
MOVJ C03824 VJ=0.78
MOVJ C03825 VJ=0.78
MOVJ C03826 VJ=0.78
MOVL C03827 V=8.0
MOVJ C03828 VJ=0.78
MOVJ C03829 VJ=0.78
MOVJ C03830 VJ=0.78
MOVL C03831 V=8.0
MOVJ C03832 VJ=0.78
MOVJ C03833 VJ=0.78
MOVJ C03834 VJ=0.78
MOVL C03835 V=8.0
MOVJ C03836 VJ=0.78
MOVJ C03837 VJ=0.78
MOVJ C03838 VJ=0.78
MOVL C03839 V=8.0
MOVJ C03840 VJ=0.78
MOVJ C03841 VJ=0.78
MOVJ C03842 VJ=0.78
MOVL C03843 V=8.0
MOVJ C03844 VJ=0.78
MOVJ C03845 VJ=0.78
MOVJ C03846 VJ=0.78
MOVL C03847 V=8.0
MOVJ C03848 VJ=0.78
MOVJ C03849 VJ=0.78
MOVJ C03850 VJ=0.78
MOVL C03851 V=8.0
MOVJ C03852 VJ=0.78
MOVJ C03853 VJ=0.78
MOVJ C03854 VJ=0.78
MOVL C03855 V=8.0
MOVJ C03856 VJ=0.78
MOVJ C03857 VJ=0.78
MOVJ C03858 VJ=0.78
MOVL C03859 V=8.0
MOVJ C03860 VJ=0.78
MOVJ C03861 VJ=0.78
MOVJ C03862 VJ=0.78
MOVL C03863 V=8.0
MOVJ C03864 VJ=0.78
MOVJ C03865 VJ=0.78
MOVJ C03866 VJ=0.78
MOVL C03867 V=8.0
MOVJ C03868 VJ=0.78
MOVJ C03869 VJ=0.78
MOVJ C03870 VJ=0.78
MOVL C03871 V=8.0
MOVJ C03872 VJ=0.78
MOVJ C03873 VJ=0.78
MOVJ C03874 VJ=0.78
MOVL C03875 V=8.0
MOVJ C03876 VJ=0.78
MOVJ C03877 VJ=0.78
MOVJ C03878 VJ=0.78
MOVL C03879 V=8.0
MOVJ C03880 VJ=0.78
MOVJ C03881 VJ=0.78
MOVJ C03882 VJ=0.78
MOVL C03883 V=8.0
MOVJ C03884 VJ=0.78
MOVJ C03885 VJ=0.78
MOVJ C03886 VJ=0.78
MOVL C03887 V=8.0
MOVJ C03888 VJ=0.78
MOVJ C03889 VJ=0.78
MOVJ C03890 VJ=0.78
MOVL C03891 V=8.0
MOVJ C03892 VJ=0.78
MOVJ C03893 VJ=0.78
MOVJ C03894 VJ=0.78
MOVL C03895 V=8.0
MOVJ C03896 VJ=0.78
MOVJ C03897 VJ=0.78
MOVJ C03898 VJ=0.78
MOVL C03899 V=8.0
MOVJ C03900 VJ=0.78
MOVJ C03901 VJ=0.78
MOVJ C03902 VJ=0.78
MOVL C03903 V=8.0
MOVJ C03904 VJ=0.78
MOVJ C03905 VJ=0.78
MOVJ C03906 VJ=0.78
MOVL C03907 V=8.0
MOVJ C03908 VJ=0.78
MOVJ C03909 VJ=0.78
MOVJ C03910 VJ=0.78
MOVL C03911 V=8.0
MOVJ C03912 VJ=0.78
MOVJ C03913 VJ=0.78
MOVJ C03914 VJ=0.78
MOVL C03915 V=8.0
MOVJ C03916 VJ=0.78
MOVJ C03917 VJ=0.78
MOVJ C03918 VJ=0.78
MOVL C03919 V=8.0
MOVJ C03920 VJ=0.78
MOVJ C03921 VJ=0.78
MOVJ C03922 VJ=0.78
MOVL C03923 V=8.0
MOVJ C03924 VJ=0.78
MOVJ C03925 VJ=0.78
MOVJ C03926 VJ=0.78
MOVL C03927 V=8.0
MOVJ C03928 VJ=0.78
MOVJ C03929 VJ=0.78
MOVJ C03930 VJ=0.78
MOVL C03931 V=8.0
MOVJ C03932 VJ=0.78
MOVJ C03933 VJ=0.78
MOVJ C03934 VJ=0.78
MOVL C03935 V=8.0
MOVJ C03936 VJ=0.78
MOVJ C03937 VJ=0.78
MOVJ C03938 VJ=0.78
MOVL C03939 V=8.0
MOVJ C03940 VJ=0.78
MOVJ C03941 VJ=0.78
MOVJ C03942 VJ=0.78
MOVL C03943 V=8.0
MOVJ C03944 VJ=0.78
MOVJ C03945 VJ=0.78
MOVJ C03946 VJ=0.78
MOVL C03947 V=8.0
MOVJ C03948 VJ=0.78
MOVJ C03949 VJ=0.78
MOVJ C03950 VJ=0.78
MOVL C03951 V=8.0
MOVJ C03952 VJ=0.78
MOVJ C03953 VJ=0.78
MOVJ C03954 VJ=0.78
MOVL C03955 V=8.0
MOVJ C03956 VJ=0.78
MOVJ C03957 VJ=0.78
MOVJ C03958 VJ=0.78
MOVL C03959 V=8.0
MOVJ C03960 VJ=0.78
MOVJ C03961 VJ=0.78
MOVJ C03962 VJ=0.78
MOVL C03963 V=8.0
MOVJ C03964 VJ=0.78
MOVJ C03965 VJ=0.78
MOVJ C03966 VJ=0.78
MOVL C03967 V=8.0
MOVJ C03968 VJ=0.78
MOVJ C03969 VJ=0.78
MOVJ C03970 VJ=0.78
MOVL C03971 V=8.0
MOVJ C03972 VJ=0.78
MOVJ C03973 VJ=0.78
MOVJ C03974 VJ=0.78
MOVL C03975 V=8.0
MOVJ C03976 VJ=0.78
MOVJ C03977 VJ=0.78
MOVJ C03978 VJ=0.78
MOVL C03979 V=8.0
MOVJ C03980 VJ=0.78
MOVJ C03981 VJ=0.78
MOVJ C03982 VJ=0.78
MOVL C03983 V=8.0
MOVJ C03984 VJ=0.78
MOVJ C03985 VJ=0.78
MOVJ C03986 VJ=0.78
MOVL C03987 V=8.0
MOVJ C03988 VJ=0.78
MOVJ C03989 VJ=0.78
MOVJ C03990 VJ=0.78
MOVL C03991 V=8.0
MOVJ C03992 VJ=0.78
MOVJ C03993 VJ=0.78
MOVJ C03994 VJ=0.78
MOVL C03995 V=8.0
MOVJ C03996 VJ=0.78
MOVJ C03997 VJ=0.78
MOVJ C03998 VJ=0.78
MOVL C03999 V=8.0
MOVJ C04000 VJ=0.78
MOVJ C04001 VJ=0.78
MOVJ C04002 VJ=0.78
MOVL C04003 V=8.0
MOVJ C04004 VJ=0.78
MOVJ C04005 VJ=0.78
MOVJ C04006 VJ=0.78
MOVL C04007 V=8.0
MOVJ C04008 VJ=0.78
MOVJ C04009 VJ=0.78
MOVJ C04010 VJ=0.78
MOVL C04011 V=8.0
MOVJ C04012 VJ=0.78
MOVJ C04013 VJ=0.78
MOVJ C04014 VJ=0.78
MOVL C04015 V=8.0
MOVJ C04016 VJ=0.78
MOVJ C04017 VJ=0.78
MOVJ C04018 VJ=0.78
MOVL C04019 V=8.0
MOVJ C04020 VJ=0.78
MOVJ C04021 VJ=0.78
MOVJ C04022 VJ=0.78
MOVL C04023 V=8.0
MOVJ C04024 VJ=0.78
MOVJ C04025 VJ=0.78
MOVJ C04026 VJ=0.78
MOVL C04027 V=8.0
MOVJ C04028 VJ=0.78
MOVJ C04029 VJ=0.78
MOVJ C04030 VJ=0.78
MOVL C04031 V=8.0
MOVJ C04032 VJ=0.78
MOVJ C04033 VJ=0.78
MOVJ C04034 VJ=0.78
MOVL C04035 V=8.0
MOVJ C04036 VJ=0.78
MOVJ C04037 VJ=0.78
MOVJ C04038 VJ=0.78
MOVL C04039 V=8.0
MOVJ C04040 VJ=0.78
END
